// TwinCAT 3 PLC project Untitled1
// ProgramVersion: 3.1.4024.0
// libraries:
//   Tc2_Standard, * (Beckhoff Automation GmbH)
//   Tc2_System, * (Beckhoff Automation GmbH)
//   Tc3_EventLogger, * (Beckhoff Automation GmbH)
//   Tc3_Module, * (Beckhoff Automation GmbH)
// project tree:
//   / PlcTask.TcTTO
//   POUs/ MAIN.TcPOU
// real-time tasks:
//   TASK PlcTask: cycle T#10ms, priority 20, ADS port 350

CONFIGURATION Untitled1
    RESOURCE PLC ON TwinCAT3
        TASK PlcTask(INTERVAL := T#10ms, PRIORITY := 20);
        PROGRAM MAIN WITH PlcTask : MAIN;
    END_RESOURCE
END_CONFIGURATION

// ---- POUs/MAIN.TcPOU
PROGRAM MAIN
VAR
	fbAlarm : FB_TcAlarm;
	fbMessage : FB_TcMessage;
	bInit : BOOL := TRUE;
	
	bRaiseAlarm: BOOL;
	bAlarmClear: BOOL;
	bAlarmConfirm: BOOL;
	bSendMessage: BOOL;
END_VAR

IF binit THEN 
	binit := FALSE;
	fbAlarm.CreateEx(stEventEntry := TC_Events.SampleEventClass.ToBeAlarm,1,0);
	fbMessage.CreateEx(stEventEntry := TC_EVENTS.SampleEventClass.ToBeMessage,0);
END_IF

IF bRaiseAlarm THEN 
	bRaiseAlarm := FALSE;
	fbAlarm.Raise(0);
END_IF

IF bAlarmClear THEN 
	bAlarmClear := FALSE;
	fbAlarm.Clear(nTimeStamp := 0, bResetConfirmation := TRUE);
END_IF

IF bAlarmConfirm THEN 
	bAlarmConfirm := FALSE;
	fbAlarm.Confirm(0);
END_IF

IF bSendMessage THEN 
	bSendMessage := FALSE;
	fbMessage.Send(0);
END_IF

END_PROGRAM
